FUNCTION_BLOCK XtsTrackStub IMPLEMENTS I_XtsTrack
VAR_INPUT
END_VAR
VAR_OUTPUT
END_VAR
VAR
	_trackLength : MC_LREAL  := 1000;
END_VAR

{warning 'add property implementation'}
PROPERTY MyOTCID : OTCID
GET
END_GET
SET
END_SET
END_PROPERTY

{warning 'add property implementation'}
PROPERTY TrackLength : MC_Lreal
GET
tracklength := _trackLength;
END_GET
END_PROPERTY

END_FUNCTION_BLOCK

(* stored: Version 1.1.0.1
   POU XtsTrackStub: Id {9bbdc397-a1f7-4a22-bd28-c8ebf47c132d}, SpecialFunc None
   Property MyOTCID: Id {82e92a1c-ecd4-4993-863a-3adb035740db}
   Get Get: Id {d8839110-2373-4ef4-848a-6531a30d1bca}
   Set Set: Id {2a4232e3-ad71-45d8-9e93-375892f77c94}
   Property TrackLength: Id {fa20ce29-545f-440e-8f6d-875dc2b61ead}
   Get Get: Id {24c356d3-cb16-44c5-8eb7-15f581e09659} *)
